TYPE ST_Assert :
STRUCT
	eAssert:		E_Assert;
	sMessage:		STRING(255);
	sType:			STRING(255);
	sData:			STRING(255);	
END_STRUCT
END_TYPE

(* stored: Version 1.1.0.1
   DUT ST_Assert: Id {8bec824b-498f-012d-1ff2-7dca2205fb5d} *)
